Staubli VAL3: ros_i_driver.dtx

public bool bFbkOverrun
public bool bMotionOverrun
public jointRx jCurrPose
mdesc mNomSpeed = {blend=off}
public num nCounter
public num nFbkPeriod = 0.032
public num nLengthB[4]
num nMotionPeriod = 0.012
public num nPosVelAccB[120]
public num nRetVal
public num nRobotIdB[4]
public num nTimeB[4]
public num nValidFieldsB[4] = 2
public sio siTcpIpFbk = {link=Socket\Feedback}
public sio siTcpIpMotion = {link=Socket\Motion}
public string sFbkTaskName = "publisher"
public string sMotionTaskName
public num nMsgTypeB[4]
public num nCommTypeB[4]
public num nReplyCodeB[4]
public RosSimpleMsg rosMsgJointFbk
  [0]
    Header header
      [0]
        num nMsgType
        num nCommType
        num nReplyCode
    Prefix prefix
      [0]
        num nLength
    Body body
      [0]
        num nData[33]
public bool bStream
public num nBytesSent
public RosSimpleMsg rosMsgJState
  [0]
    Header header
      [0]
        num nMsgType
        num nCommType
        num nReplyCode
    Prefix prefix
      [0]
        num nLength
    Body body
      [0]
        num nData[11]
public num nSeqB[4]
public num nPosB[40]
public num nDeg2Rad
